(* CODESYS project %PV%PERSIVARS.xml

Project tree, tasks and I/O mapping:
  global variables PERSIVARS
*)

// PERSIVARS
{attribute 'qualified_only'}
VAR_GLOBAL PERSISTENT RETAIN
	test1: BOOL;
	test2: INT;
END_VAR
